FUNCTION_BLOCK FB_Observer_LREAL_ EXTENDS TcBase.FB_Observer_LREAL
VAR_INPUT
END_VAR
VAR_OUTPUT
END_VAR
VAR
END_VAR

PROPERTY nUpdateCounter : UDINT
GET
nUpdateCounter := THIS^._nUpdateCounter;
END_GET
END_PROPERTY

END_FUNCTION_BLOCK

(* stored: Version 1.1.0.1, ProductVersion 3.1.4024.12
   POU FB_Observer_LREAL_: Id {b8192a2c-e2e7-4cdb-9005-1d4ba8a7cd61}, SpecialFunc None
   Property nUpdateCounter: Id {0a2114c8-39b2-4fb4-88dc-6d5a6f2b8382}
   Get Get: Id {c1db33dc-503c-495b-8bf7-fad580576830} *)
